(* PLC project actuator, TNI-Software ControlBuild 4.00.17 *)
(* stored: creationDateTime 2005-06-20T11:53:06-01:00 *)

FUNCTION_BLOCK cmd_equipment_library.actuator
  VAR_INPUT  (* CB.group=Modes CB.kind=inputVars *)
    autoMode : BOOL := false;  (* CB.mnemonicPatternPropertyName=<SY>_AUTO_<NU> CB.libelle=Automatic mode *)
    manualMode : BOOL := false;  (* CB.mnemonicPatternPropertyName=<SY>_MANU_<NU> CB.libelle=Manual mode *)
  END_VAR
  VAR_INPUT  (* CB.group=Commands CB.kind=inputVars *)
    autoWorkCmd : BOOL := false;  (* CB.mnemonicPatternPropertyName=<SY>_CMDFWAUTO_<NU> CB.libelle=Automatic work command to the valve *)
    autoRestCmd : BOOL := false;  (* CB.mnemonicPatternPropertyName=<SY>_CMDSAUTO_<NU> CB.libelle=Automatic rest command to the valve *)
  END_VAR
  VAR_INPUT  (* CB.group=PushButtons CB.kind=inputVars *)
    valveWorkPB : BOOL := false;  (* CB.mnemonicPatternPropertyName=<SY>_BPFW_<NU> CB.libelle=Valve work pushbutton *)
    valveRestPB : BOOL := false;  (* CB.mnemonicPatternPropertyName=<SY>_BPS_<NU> CB.libelle=Valve rest pushbutton *)
  END_VAR
  VAR_INPUT  (* CB.group=Sensors CB.kind=inputVars *)
    outletSensor : BOOL := false;  (* CB.libelle=Outlet sensor *)
    inletSensor : BOOL := false;  (* CB.libelle=Inlet sensor *)
  END_VAR
  VAR_INPUT  (* CB.kind=inputVars *)
    generalFault : BOOL := false;  (* CB.mnemonicPatternPropertyName=<SY>_DEF_<NU> CB.libelle=General fault of the jack *)
  END_VAR
  VAR_OUTPUT  (* CB.group=Orders CB.kind=outputVars *)
    workCmd : BOOL := false;  (* CB.mnemonicPatternPropertyName=workCmd<SY><NU> CB.libelle=Work command to the valve *)
    restCmd : BOOL := false;  (* CB.mnemonicPatternPropertyName=restCmd<SY><NU> CB.libelle=Rest command to the valve *)
  END_VAR

(* LD diagram, written out as Structured Text *)
1:
workCmd := (autoMode AND (autoWorkCmd OR workCmd) AND NOT autoRestCmd OR manualMode AND valveWorkPB AND NOT valveRestPB OR manualMode AND workCmd) AND NOT outletSensor AND NOT generalFault;
2:
restCmd := (autoMode AND (autoRestCmd OR restCmd) AND NOT autoWorkCmd OR manualMode AND valveRestPB AND NOT valveWorkPB OR manualMode AND restCmd) AND NOT inletSensor AND NOT generalFault;
END_FUNCTION_BLOCK
